INTERFACE IPLCopenCaller EXTENDS IPLCopenCall

PROPERTY Busy : BOOL
GET
END_GET
END_PROPERTY

PROPERTY Command : IPLCopenCommand
GET
END_GET
SET
END_SET
END_PROPERTY

PROPERTY CommandAborted : BOOL
GET
END_GET
END_PROPERTY

PROPERTY Done : BOOL
GET
END_GET
END_PROPERTY

PROPERTY Error : BOOL
GET
END_GET
END_PROPERTY

PROPERTY Execute : BOOL
GET
END_GET
SET
END_SET
END_PROPERTY

PROPERTY Fallback : PLCopenStatusBase
GET
END_GET
SET
END_SET
END_PROPERTY

METHOD ResetStatus : BOOL
END_METHOD

END_INTERFACE

(* stored: Version 1.1.0.1
   Itf IPLCopenCaller: Id {3539bad0-84c7-0f02-0e2d-9dcc4fb33c22}
   Property Busy: Id {35f172e6-8886-0779-260d-da1cf511c014}
   Get Get: Id {d75c6d1b-1de8-03cb-154b-c5ab60116087}
   Property Command: Id {e0f4faf6-71bc-0e9d-1a78-ded425fad3b8}
   Get Get: Id {dbe69e9e-563b-07a1-27d8-f05d334de5f1}
   Set Set: Id {6d722569-e222-0e6b-0eb1-366ee5fc6131}
   Property CommandAborted: Id {8a5376e7-846f-0d1e-33f5-620b908f238f}
   Get Get: Id {16149f9a-c344-00ce-34b1-ccb943f2a19e}
   Property Done: Id {be443404-9511-070a-0351-40b4b4cbaa97}
   Get Get: Id {0f2ac159-ad36-05c1-1666-48553ef247d0}
   Property Error: Id {ea7ccb85-0051-06fa-360a-62883651b384}
   Get Get: Id {d5be0bf8-5ed8-022b-368d-d4421f994fbb}
   Property Execute: Id {b483299d-2a67-013f-29f3-98c9269ee934}
   Get Get: Id {4f130ee4-ef52-0dc1-3a0f-ea31e9042a4f}
   Set Set: Id {bdc8426a-c2c7-0ce2-23a9-bea63fb21cf1}
   Property Fallback: Id {1364c025-da75-018e-146b-189874eb68d2}
   Get Get: Id {a90463fe-4a50-0b76-199d-7bc517e6cf8f}
   Set Set: Id {742930a6-c0dd-0605-3185-310e54a04a23}
   Method ResetStatus: Id {81b3fc3a-1372-0b12-38fe-bd388ba1f607} *)
